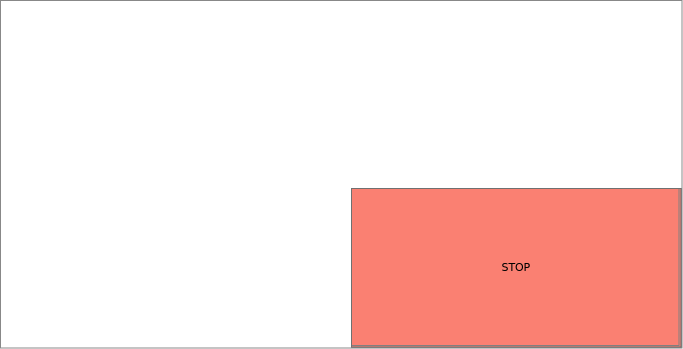
VISUALIZATION Visualization  // 683x349
    Button (351,188 330x159), "STOP", colour toggle: GVL.StopALL
        toggle GVL.StopALL
END_VISUALIZATION

(* stored: Version 1.1.0.1, ProductVersion 3.1.4024.2
   Visu Visualization: Id {cc4fa22e-8baa-4d95-9844-dc806d2abdcd} *)
